// TIA Portal V19 export
TYPE "HMI_Preset"
// stored: Access Published
   STRUCT
      Button : Bool;   // Pulsante HMI che lancia il comando di preset
      Value : LReal;   // Valore di preset
      Feedback : LReal;   // Valore di ritorno se = Value allora l'operazione è stata eseguita
   END_STRUCT;
END_TYPE
